FUNCTION_BLOCK EM_Transport IMPLEMENTS  ITF_EM_Transport, ITF_PackML

VAR
	fb_mem : STRUCT_EM_Transport;
	
	Motor		: CM_Motor;
	Sensor		: CM_Sensor;
END_VAR

(*
$$$$$$$$\                                                                   $$\       $$$$$$$$\                     $$\                                         $$\                     
$$  _____|                                                                  $$ |      $$  _____|                    \__|                                        \__|                    
$$ |   $$$$$$\   $$$$$$\  $$$$$$$\  $$\  $$\  $$\  $$$$$$\   $$$$$$\   $$$$$$$ |      $$ |      $$$$$$$\   $$$$$$\  $$\ $$$$$$$\   $$$$$$\   $$$$$$\   $$$$$$\  $$\ $$$$$$$\   $$$$$$\  
$$$$$\ \____$$\ $$  __$$\ $$  __$$\ $$ | $$ | $$ |$$  __$$\ $$  __$$\ $$  __$$ |      $$$$$\    $$  __$$\ $$  __$$\ $$ |$$  __$$\ $$  __$$\ $$  __$$\ $$  __$$\ $$ |$$  __$$\ $$  __$$\ 
$$  __|$$$$$$$ |$$ |  \__|$$ |  $$ |$$ | $$ | $$ |$$ /  $$ |$$ /  $$ |$$ /  $$ |      $$  __|   $$ |  $$ |$$ /  $$ |$$ |$$ |  $$ |$$$$$$$$ |$$$$$$$$ |$$ |  \__|$$ |$$ |  $$ |$$ /  $$ |
$$ |  $$  __$$ |$$ |      $$ |  $$ |$$ | $$ | $$ |$$ |  $$ |$$ |  $$ |$$ |  $$ |      $$ |      $$ |  $$ |$$ |  $$ |$$ |$$ |  $$ |$$   ____|$$   ____|$$ |      $$ |$$ |  $$ |$$ |  $$ |
$$ |  \$$$$$$$ |$$ |      $$ |  $$ |\$$$$$\$$$$  |\$$$$$$  |\$$$$$$  |\$$$$$$$ |      $$$$$$$$\ $$ |  $$ |\$$$$$$$ |$$ |$$ |  $$ |\$$$$$$$\ \$$$$$$$\ $$ |      $$ |$$ |  $$ |\$$$$$$$ |
\__|   \_______|\__|      \__|  \__| \_____\____/  \______/  \______/  \_______|      \________|\__|  \__| \____$$ |\__|\__|  \__| \_______| \_______|\__|      \__|\__|  \__| \____$$ |
                                                                                                          $$\   $$ |                                                          $$\   $$ |
                                                                                                          \$$$$$$  |                                                          \$$$$$$  |
                                                                                                           \______/                                                            \______/ 
*)
//********************************Initiating***********************************
fb_mem.STS.State := PackML_StateMachine(State			:= fb_mem.STS.State,
										Start           := fb_mem.CS.Start,
										Stop            := fb_mem.CS.Stop,
										Reset           := fb_mem.CS.Reset,
										Abort           := fb_mem.CS.Abort,
										Clear           := fb_mem.CS.Clear,
										UnSuspend       := fb_mem.CS.UnSuspend,
										Suspend         := fb_mem.CS.Suspend,
										UnHold          := fb_mem.CS.UnHold,
										Hold            := fb_mem.CS.Hold,
										Starting_SC     := fb_mem.STS.Starting_SC,
										Execute_SC      := fb_mem.STS.Execute_SC,
										Resetting_SC    := fb_mem.STS.Resetting_SC,
										Holding_SC      := fb_mem.STS.Holding_SC,
										Unholding_SC    := fb_mem.STS.Unholding_SC,
										Suspending_SC   := fb_mem.STS.Suspending_SC,
										Unsuspending_SC := fb_mem.STS.Unsuspending_SC,
										Aborting_SC     := fb_mem.STS.Aborting_SC,
										Clearing_SC     := fb_mem.STS.Clearing_SC,
										Stopping_SC     := fb_mem.STS.Stopping_SC);
//********************************Init***********************************
Motor();
Sensor();
										
//********************************ZEROING***********************************		
(*							
fb_mem.STS.Auto 			:= FALSE;
fb_mem.STS.Manueel 			:= FALSE;
fb_mem.STS.Starting_SC 		:= FALSE;
fb_mem.STS.Execute_SC 		:= FALSE;
fb_mem.STS.Resetting_SC 	:= FALSE;
fb_mem.STS.Holding_SC 		:= FALSE;
fb_mem.STS.Unholding_SC 	:= FALSE;
fb_mem.STS.Suspending_SC 	:= FALSE;
fb_mem.STS.Unsuspending_SC 	:= FALSE;
fb_mem.STS.Aborting_SC 		:= FALSE;
fb_mem.STS.Clearing_SC 		:= FALSE;
fb_mem.STS.Stopping_SC 		:= FALSE;
fb_mem.STS.Completing_SC 	:= FALSE;
*)

//********************************Auto manual logic***********************************
IF fb_mem.CS.Auto THEN
	fb_mem.STS.Auto := TRUE;
	ELSE
		fb_mem.STS.Auto := FALSE;
END_IF

IF fb_mem.CS.Manueel THEN
	fb_mem.STS.Manueel := TRUE;
	ELSE
		fb_mem.STS.Manueel := FALSE;
END_IF

//********************************Exeptionhandling***********************************

//********************************Action case***********************************
CASE fb_mem.STS.State OF
	E_State_PackML.IDLE 			: 
		//Do nothing
	E_State_PackML.STARTING 		:
		Motor.Start();
		IF Motor.State = E_State_PackML.EXECUTE THEN
			fb_mem.STS.Starting_SC 		:= TRUE;	
		END_IF
	E_State_PackML.EXECUTE 			: 
		//Do nothing
	E_State_PackML.COMPLETE 		:
		Motor.Reset();
		IF Motor.State = E_State_PackML.RESETTING THEN
			fb_mem.STS.Completing_SC := TRUE;
		END_IF
	E_State_PackML.RESETTING 		:
		FB_init(0,0);
		Motor.FB_init(0,0);
		IF Motor.State = E_State_PackML.IDLE THEN
			fb_mem.STS.Resetting_SC 	:= TRUE;
		END_IF
	E_State_PackML.HOLDING 			:
		Motor.Stop();
		IF Motor.State = E_State_PackML.STOPPED THEN
			fb_mem.STS.Unholding_SC		:= TRUE;
		END_IF
	E_State_PackML.HELD 			:
		//Do nothing
	E_State_PackML.UNHOLDING 		:
		Motor.Reset();
		Motor.Reset();
		IF Motor.State = E_State_PackML.EXECUTE THEN
			fb_mem.STS.Unholding_SC		:= TRUE;
		END_IF
	E_State_PackML.SUSPENDING 		:
		Motor.Stop();
		IF Motor.State = E_State_PackML.STOPPED THEN
			fb_mem.STS.Suspending_SC 	:= TRUE;
		END_IF
	E_State_PackML.SUSPENDED 		:
		//Do nothing
	E_State_PackML.UNSUSPENDING 	:
		Motor.Reset();
		Motor.Reset();
		IF Motor.State = E_State_PackML.EXECUTE THEN
			fb_mem.CS.Unsuspend 		:= TRUE;
		END_IF
	E_State_PackML.ABORTING			:
		Motor.Abort();
		IF Motor.State = E_State_PackML.ABORTED THEN
			fb_mem.STS.Aborting_SC 		:= TRUE;
		END_IF
	E_State_PackML.ABORTED			:
		//Do nothing
	E_State_PackML.CLEARING 		:
		Motor.Clear();
		IF Motor.State = E_State_PackML.STOPPED THEN
			fb_mem.STS.Clearing_SC 		:= TRUE;
		END_IF
	E_State_PackML.STOPPING 		:
		IF Motor.State = E_State_PackML.STOPPED THEN
			fb_mem.STS.Stopping_SC 		:= TRUE;
		END_IF
	E_State_PackML.STOPPED 			:
		//Do nothing
END_CASE



//********************************ZEROING***********************************
//Control Signals 
(*
fb_mem.CS.Auto            := FALSE;
fb_mem.CS.Manueel         := FALSE;
fb_mem.CS.Start           := FALSE;
fb_mem.CS.Stop            := FALSE;
fb_mem.CS.Reset           := FALSE;
fb_mem.CS.Abort           := FALSE;
fb_mem.CS.Clear           := FALSE;
fb_mem.CS.UnSuspend       := FALSE;
fb_mem.CS.Suspend         := FALSE;
fb_mem.CS.UnHold          := FALSE;
fb_mem.CS.Hold            := FALSE;
*)

{warning 'add method implementation '}
METHOD Abort : BOOL
fb_mem.CS.Abort := TRUE;
END_METHOD

METHOD Aborting_SC : BOOL
VAR_INPUT
END_VAR
fb_mem.STS.Aborting_SC := TRUE;
END_METHOD

{warning 'add method implementation '}
METHOD Auto : BOOL
fb_mem.CS.Auto := TRUE;
fb_mem.CS.Manueel := FALSE;

Auto := fb_mem.STS.Auto;
END_METHOD

{warning 'add method implementation '}
METHOD Clear : BOOL
fb_mem.CS.Clear := TRUE;
END_METHOD

METHOD Clearing_SC : BOOL
VAR_INPUT
END_VAR
fb_mem.STS.Clearing_SC := TRUE;
END_METHOD

METHOD Completing_SC : BOOL
VAR_INPUT
END_VAR
fb_mem.STS.Completing_SC := TRUE;
END_METHOD

METHOD Execute_SC : BOOL
VAR_INPUT
END_VAR
fb_mem.STS.Execute_SC := TRUE;
END_METHOD

{warning 'add method implementation '}
METHOD FB_init : BOOL
VAR_INPUT
	(* if TRUE, the retain variables are initialized (warm start / cold start)*)
	bInitRetains	: BOOL;
	(* if TRUE, the instance afterwards gets moved into the copy code (online change)*)
	bInCopyCode	: BOOL;
END_VAR
END_METHOD

{warning 'add method implementation '}
METHOD Hold : BOOL
fb_mem.CS.Hold := TRUE;
END_METHOD

METHOD Holding_SC : BOOL
VAR_INPUT
END_VAR
fb_mem.STS.Holding_SC := TRUE;
END_METHOD

{warning 'add method implementation '}
METHOD Manueel : BOOL
fb_mem.CS.Manueel := TRUE;
fb_mem.CS.Auto := FALSE;

Manueel := fb_mem.STS.Manueel;
END_METHOD

{warning 'add method implementation '}
METHOD Reset : BOOL
fb_mem.CS.Reset := TRUE;
END_METHOD

METHOD Resetting_SC : BOOL
VAR_INPUT
END_VAR
fb_mem.STS.Resetting_SC := TRUE;
END_METHOD

{warning 'add property implementation'}
PROPERTY RPM : INT
GET
END_GET
SET
END_SET
END_PROPERTY

{warning 'add method implementation '}
METHOD Start : BOOL
fb_mem.CS.Start := TRUE;
END_METHOD

METHOD Starting_SC : BOOL
VAR_INPUT
END_VAR
fb_mem.STS.Starting_SC := TRUE;
END_METHOD

{warning 'add property implementation'}
PROPERTY State : E_State_PackML
GET
State := fb_mem.STS.State;
END_GET
END_PROPERTY

{warning 'add method implementation '}
METHOD Stop : BOOL
fb_mem.CS.Stop := TRUE;
END_METHOD

METHOD Stopping_SC : BOOL
VAR_INPUT
END_VAR
fb_mem.STS.Stopping_SC := TRUE;
END_METHOD

{warning 'add method implementation '}
METHOD Suspend : BOOL
fb_mem.CS.Suspend := TRUE;
END_METHOD

METHOD Suspending_SC : BOOL
VAR_INPUT
END_VAR
fb_mem.STS.Suspending_SC := TRUE;
END_METHOD

{warning 'add property implementation'}
PROPERTY Tag : STRING
GET
Tag := fb_mem.STS.Tag;
END_GET
END_PROPERTY

{warning 'add method implementation '}
METHOD Unhold : BOOL
fb_mem.CS.Unhold := TRUE;
END_METHOD

METHOD Unholding_SC : BOOL
VAR_INPUT
END_VAR
fb_mem.STS.Unholding_SC := TRUE;
END_METHOD

{warning 'add method implementation '}
METHOD Unsuspend : BOOL
fb_mem.CS.Unsuspend := TRUE;
END_METHOD

METHOD Unsuspending_SC : BOOL
VAR_INPUT
END_VAR
fb_mem.STS.Unsuspending_SC := TRUE;
END_METHOD

{warning 'add method implementation '}
METHOD ZeroAllVar : BOOL
END_METHOD

END_FUNCTION_BLOCK

(* stored: Version 1.1.0.1, ProductVersion 3.1.4024.12
   POU EM_Transport: Id {b4839b78-b43e-43c9-b2a5-dfab2150ed70}, SpecialFunc None
   Folder Methods: Id {60ae86de-bafc-440d-bc9f-96901a1f7546}
   Folder Properties: Id {8dc97ebe-3ace-4fdf-a1ba-2a3cf702ba1f}
   Method Abort: Id {bbfdf4eb-6570-4a13-a46b-57e480ef120b}
   Method Aborting_SC: Id {8fc50448-f1f2-4e0c-8a72-b9cb3e36567e}
   Method Auto: Id {0e7aef80-4c85-478b-a934-c85e954995c2}
   Method Clear: Id {4bc6a9ab-0b4b-4eca-988f-8ccb82ec9a45}
   Method Clearing_SC: Id {b148045c-cd6e-4b03-9f89-a120c7e9b391}
   Method Completing_SC: Id {5a776b9f-0e5f-4a47-816e-8d498528bb16}
   Method Execute_SC: Id {e65b1cb9-fa51-46f9-929e-dac6af8386bc}
   Method FB_init: Id {fef1f4a5-7c17-426e-92ad-ed7f8ff1b0d0}
   Method Hold: Id {f3cd4036-7e0c-4476-9fe9-610efdb989cd}
   Method Holding_SC: Id {bf48253a-7f00-433f-bd8e-dac1dd77a465}
   Method Manueel: Id {ede4cda6-f1de-40d8-8a49-f05d845e9d0c}
   Method Reset: Id {9693ed28-985a-456a-9662-9dcebab0097c}
   Method Resetting_SC: Id {8d281091-fe44-4095-8a17-7953d2fa6810}
   Property RPM: Id {d26f9484-70ed-43f2-858c-07c0b43837bd}
   Get Get: Id {56fdee3c-d30a-45a6-bc9a-95697aff9df6}
   Set Set: Id {143a8ab9-f354-4ba7-88c1-f0978b1d945a}
   Method Start: Id {1baf41d7-4b14-4001-bcc1-77b5d5415aba}
   Method Starting_SC: Id {8f4eb6a6-b488-4fd3-81e5-f929a091d1b3}
   Property State: Id {046af506-8cf0-46af-a509-5569994c5df0}
   Get Get: Id {027b1301-0c1f-44f4-a2eb-518122c4d3ed}
   Method Stop: Id {14c6723a-9d9f-4490-91db-62f5947b6f7d}
   Method Stopping_SC: Id {0e917c7d-c2c6-4de0-9723-1f2c1a7b0b0e}
   Method Suspend: Id {aa09acce-0447-4fc2-8ad3-1029f3d40615}
   Method Suspending_SC: Id {5b7ceb42-39ff-4e22-aaf0-2e85b78849ff}
   Property Tag: Id {7b2c485a-3821-43e3-83a2-c27ca1c63059}
   Get Get: Id {5aa24341-14dd-4f8f-bca1-bc219fc01e1b}
   Method Unhold: Id {3167d149-a93f-4223-8d89-c088f2d59da7}
   Method Unholding_SC: Id {0a22e87d-935a-479d-94e5-839f753e0237}
   Method Unsuspend: Id {d3f7206f-77e9-492e-9706-92490e1bd093}
   Method Unsuspending_SC: Id {f3cb3639-112b-4440-895c-62ae94513958}
   Method ZeroAllVar: Id {5e234a29-db91-4e63-8d3f-61453402a21d} *)
